PROGRAM PRG_AtTransfer02
VAR
	intnFBSensor : FB_Sensors;
END_VAR

intnFBSensor (
	iSensor := At_Transfer_2,
	iTimeToActuateSensor := 0,
);

END_PROGRAM

(* stored: Version 1.1.0.1
   POU PRG_AtTransfer02: Id {5c776c09-163c-4b49-9c8d-e338b978bfa8}, SpecialFunc None *)
